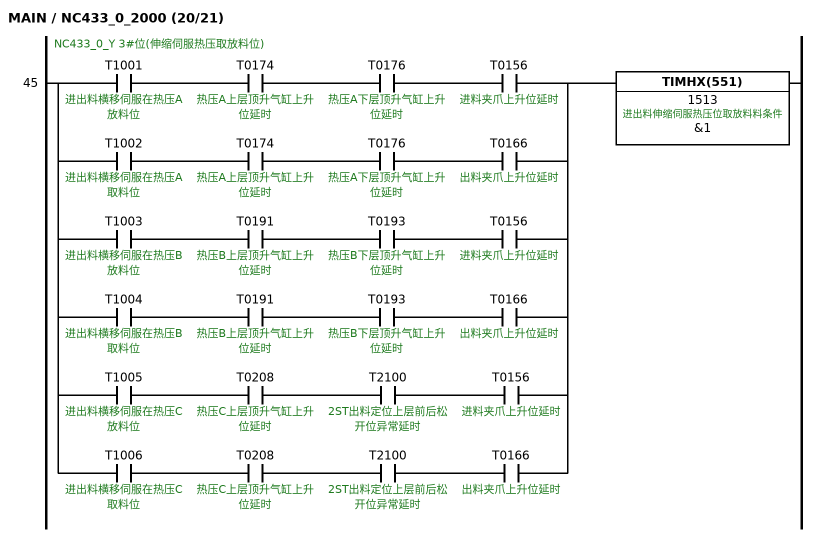
; [picture p24: MAIN / NC433_0_2000, rungs 45-45]
; rung 45: NC433_0_Y 3#位(伸缩伺服热压取放料位)
LD T1001  ; 进出料横移伺服在热压A放料位
AND T0174  ; 热压A上层顶升气缸上升位延时
AND T0176  ; 热压A下层顶升气缸上升位延时
AND T0156  ; 进料夹爪上升位延时
LD T1002  ; 进出料横移伺服在热压A取料位
AND T0174  ; 热压A上层顶升气缸上升位延时
AND T0176  ; 热压A下层顶升气缸上升位延时
AND T0166  ; 出料夹爪上升位延时
ORLD
LD T1003  ; 进出料横移伺服在热压B放料位
AND T0191  ; 热压B上层顶升气缸上升位延时
AND T0193  ; 热压B下层顶升气缸上升位延时
AND T0156  ; 进料夹爪上升位延时
ORLD
LD T1004  ; 进出料横移伺服在热压B取料位
AND T0191  ; 热压B上层顶升气缸上升位延时
AND T0193  ; 热压B下层顶升气缸上升位延时
AND T0166  ; 出料夹爪上升位延时
ORLD
LD T1005  ; 进出料横移伺服在热压C放料位
AND T0208  ; 热压C上层顶升气缸上升位延时
AND T2100  ; 2ST出料定位上层前后松开位异常延时
AND T0156  ; 进料夹爪上升位延时
ORLD
LD T1006  ; 进出料横移伺服在热压C取料位
AND T0208  ; 热压C上层顶升气缸上升位延时
AND T2100  ; 2ST出料定位上层前后松开位异常延时
AND T0166  ; 出料夹爪上升位延时
ORLD
TIMHX(551) 1513 &1  ; 进出料伸缩伺服热压位取放料料条件

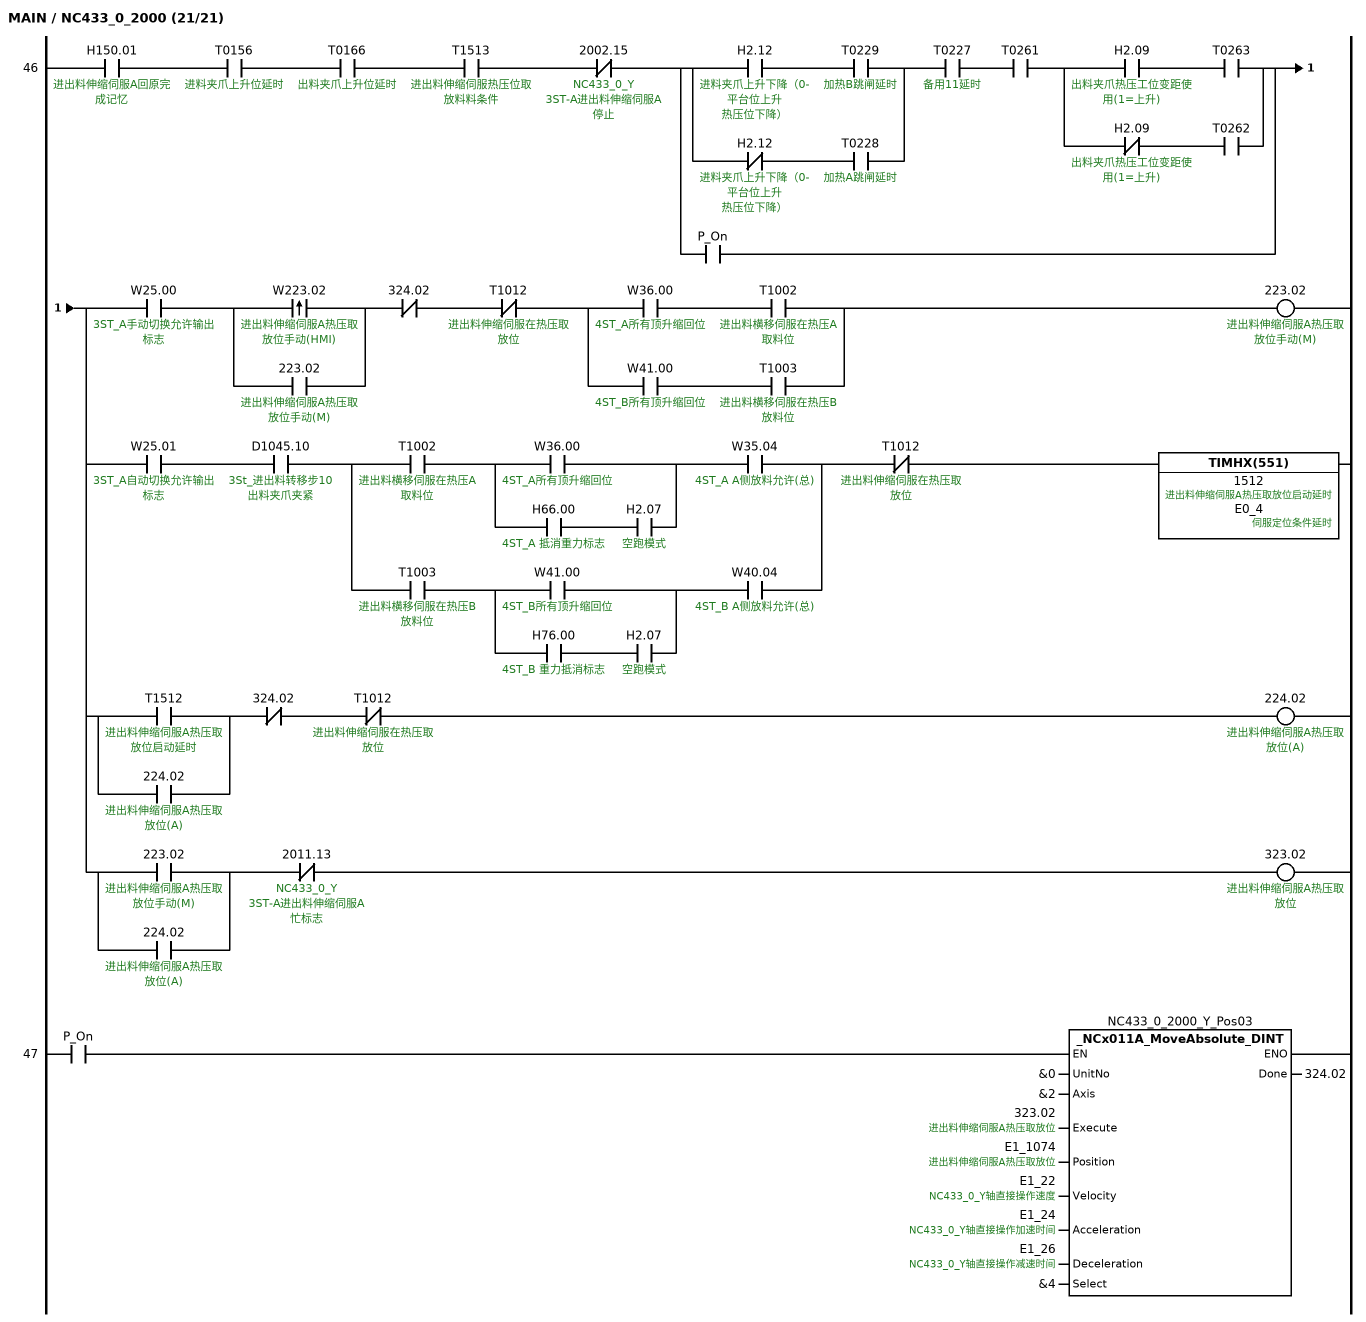
; rung 46
LD H150.01  ; 进出料伸缩伺服A回原完成记忆
AND T0156  ; 进料夹爪上升位延时
AND T0166  ; 出料夹爪上升位延时
AND T1513  ; 进出料伸缩伺服热压位取放料料条件
ANDNOT 2002.15  ; NC433_0_Y 3ST-A进出料伸缩伺服A停止
LD H2.12  ; 进料夹爪上升下降（0-平台位上升  热压位下降）
AND T0229  ; 加热B跳闸延时
LDNOT H2.12  ; 进料夹爪上升下降（0-平台位上升  热压位下降）
AND T0228  ; 加热A跳闸延时
ORLD
AND T0227  ; 备用11延时
AND T0261
LD H2.09  ; 出料夹爪热压工位变距使用(1=上升)
AND T0263
LDNOT H2.09  ; 出料夹爪热压工位变距使用(1=上升)
AND T0262
ORLD
ANDLD
OR P_On
ANDLD
OUT TR0
AND W25.00  ; 3ST_A手动切换允许输出标志
@LD W223.02  ; 进出料伸缩伺服A热压取放位手动(HMI)
OR 223.02  ; 进出料伸缩伺服A热压取放位手动(M)
ANDLD
ANDNOT 324.02
ANDNOT T1012  ; 进出料伸缩伺服在热压取放位
LD W36.00  ; 4ST_A所有顶升缩回位
AND T1002  ; 进出料横移伺服在热压A取料位
LD W41.00  ; 4ST_B所有顶升缩回位
AND T1003  ; 进出料横移伺服在热压B放料位
ORLD
ANDLD
OUT 223.02  ; 进出料伸缩伺服A热压取放位手动(M)
LD TR0
AND W25.01  ; 3ST_A自动切换允许输出标志
AND D1045.10  ; 3St_进出料转移步10 出料夹爪夹紧
LD T1002  ; 进出料横移伺服在热压A取料位
LD W36.00  ; 4ST_A所有顶升缩回位
LD H66.00  ; 4ST_A 抵消重力标志
AND H2.07  ; 空跑模式
ORLD
ANDLD
AND W35.04  ; 4ST_A A侧放料允许(总)
LD T1003  ; 进出料横移伺服在热压B放料位
LD W41.00  ; 4ST_B所有顶升缩回位
LD H76.00  ; 4ST_B 重力抵消标志
AND H2.07  ; 空跑模式
ORLD
ANDLD
AND W40.04  ; 4ST_B A侧放料允许(总)
ORLD
ANDLD
ANDNOT T1012  ; 进出料伸缩伺服在热压取放位
TIMHX(551) 1512 E0_4  ; 伺服定位条件延时, 进出料伸缩伺服A热压取放位启动延时
LD TR0
LD T1512  ; 进出料伸缩伺服A热压取放位启动延时
OR 224.02  ; 进出料伸缩伺服A热压取放位(A)
ANDLD
ANDNOT 324.02
ANDNOT T1012  ; 进出料伸缩伺服在热压取放位
OUT 224.02  ; 进出料伸缩伺服A热压取放位(A)
LD TR0
LD 223.02  ; 进出料伸缩伺服A热压取放位手动(M)
OR 224.02  ; 进出料伸缩伺服A热压取放位(A)
ANDLD
ANDNOT 2011.13  ; NC433_0_Y 3ST-A进出料伸缩伺服A忙标志
OUT 323.02  ; 进出料伸缩伺服A热压取放位
; rung 47
LD P_On
CALL NC433_0_2000_Y_Pos03 : _NCx011A_MoveAbsolute_DINT (UnitNo := &0, Axis := &2, Execute := 323.02, Position := E1_1074, Velocity := E1_22, Acceleration := E1_24, Deceleration := E1_26, Select := &4, Done => 324.02)  ; 进出料伸缩伺服A热压取放位, NC433_0_Y轴直接操作速度, NC433_0_Y轴直接操作加速时间, NC433_0_Y轴直接操作减速时间

### Section 主副PLC交互

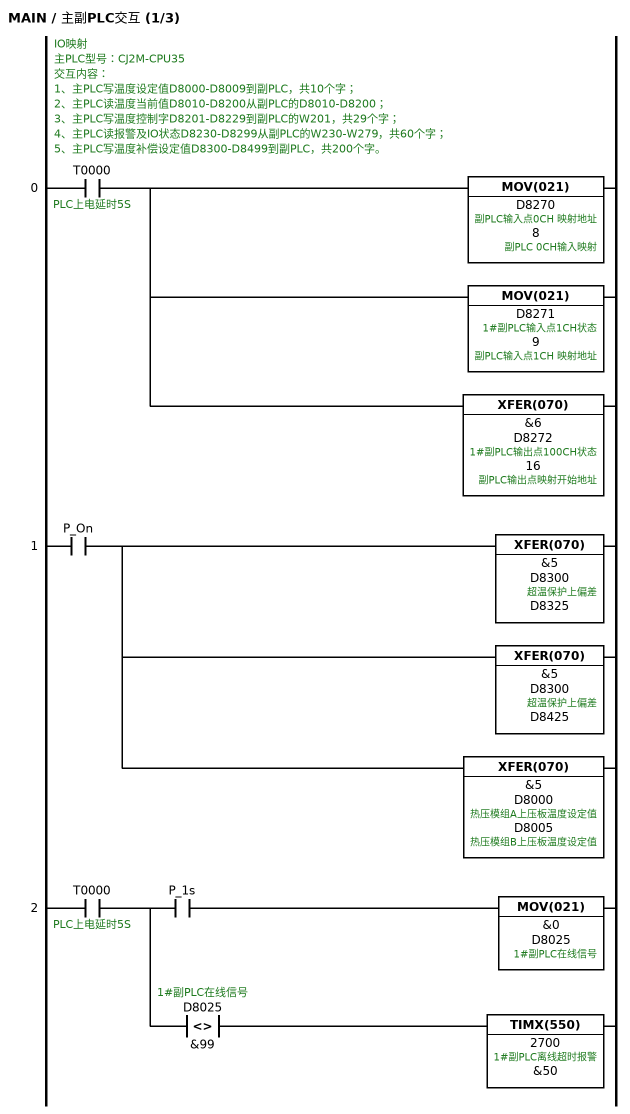
; rung 0: IO映射 / 主PLC型号：CJ2M-CPU35 / 交互内容： / 1、主PLC写温度设定值D8000-D8009到副PLC，共10个字； / 2、主PLC读温度当前值D8010-D8200从副PLC的D8010-D8200； / 3、主PLC写温度控制字D8201-D8229到副PLC的W201，共29个字； / 4、主PLC读报警及IO状态D8230-D8299从副PLC的W230-W279，共60个字； / 5、主PLC写温度补偿设定值D8300-D8499到副PLC，共200个字。
LD T0000  ; PLC上电延时5S
MOV(021) D8270 8  ; 副PLC输入点0CH 映射地址, 副PLC 0CH输入映射
MOV(021) D8271 9  ; 1#副PLC输入点1CH状态, 副PLC输入点1CH 映射地址
XFER(070) &6 D8272 16  ; 1#副PLC输出点100CH状态, 副PLC输出点映射开始地址
; rung 1
LD P_On
XFER(070) &5 D8300 D8325  ; 超温保护上偏差
XFER(070) &5 D8300 D8425  ; 超温保护上偏差
XFER(070) &5 D8000 D8005  ; 热压模组A上压板温度设定值, 热压模组B上压板温度设定值
; rung 2
LD T0000  ; PLC上电延时5S
OUT TR0
AND P_1s
MOV(021) &0 D8025  ; 1#副PLC在线信号
LD TR0
AND<>(305) D8025 &99  ; 1#副PLC在线信号
TIMX(550) 2700 &50  ; 1#副PLC离线超时报警

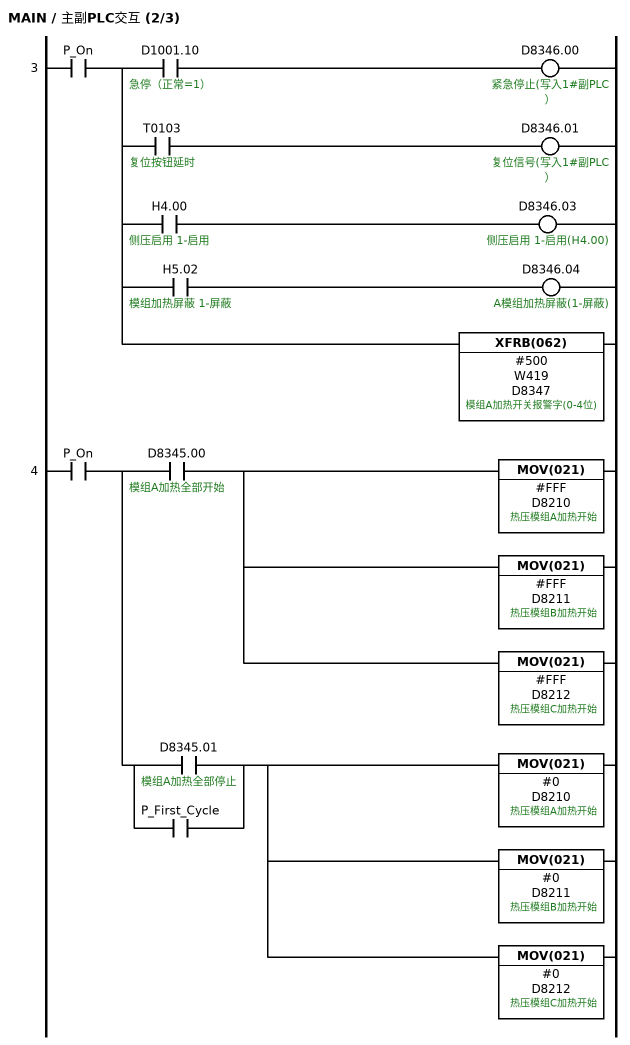
; rung 3
LD P_On
OUT TR0
AND D1001.10  ; 急停（正常=1）
OUT D8346.00  ; 紧急停止(写入1#副PLC）
LD TR0
AND T0103  ; 复位按钮延时
OUT D8346.01  ; 复位信号(写入1#副PLC）
LD TR0
AND H4.00  ; 侧压启用 1-启用
OUT D8346.03  ; 侧压启用 1-启用(H4.00)
LD TR0
AND H5.02  ; 模组加热屏蔽 1-屏蔽
OUT D8346.04  ; A模组加热屏蔽(1-屏蔽)
LD TR0
XFRB(062) #500 W419 D8347  ; 模组A加热开关报警字(0-4位)
; rung 4
LD P_On
OUT TR0
AND D8345.00  ; 模组A加热全部开始
MOV(021) #FFF D8210  ; 热压模组A加热开始
MOV(021) #FFF D8211  ; 热压模组B加热开始
MOV(021) #FFF D8212  ; 热压模组C加热开始
LD TR0
LD D8345.01  ; 模组A加热全部停止
OR P_First_Cycle
ANDLD
MOV(021) #0 D8210  ; 热压模组A加热开始
MOV(021) #0 D8211  ; 热压模组B加热开始
MOV(021) #0 D8212  ; 热压模组C加热开始

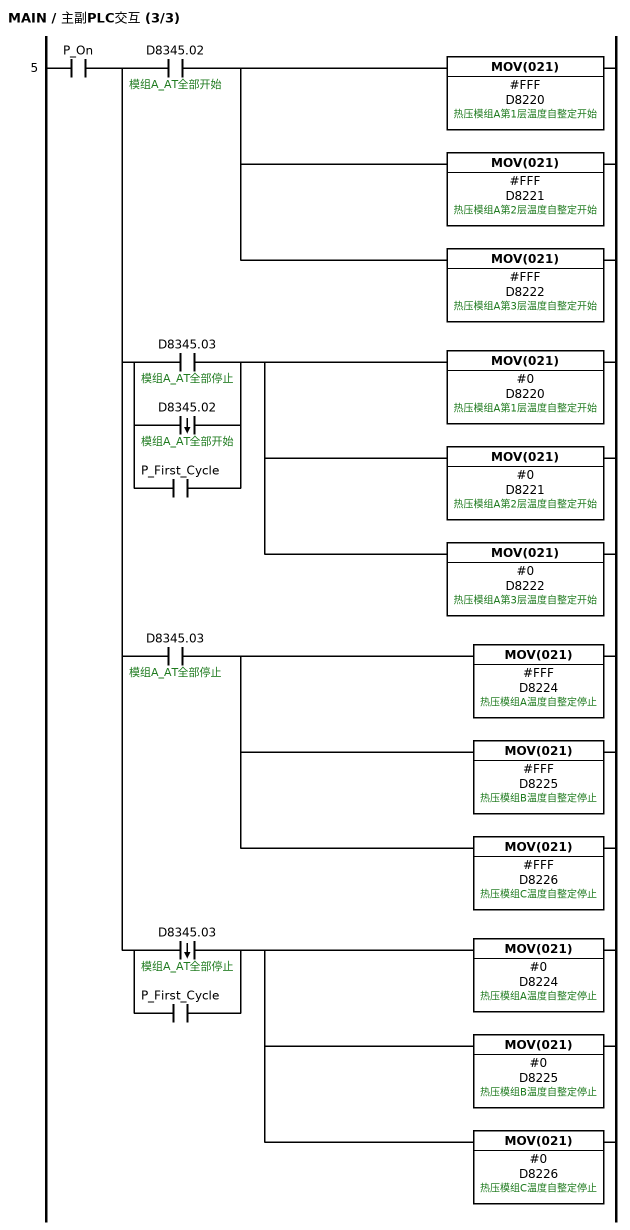
; rung 5
LD P_On
OUT TR0
AND D8345.02  ; 模组A_AT全部开始
MOV(021) #FFF D8220  ; 热压模组A第1层温度自整定开始
MOV(021) #FFF D8221  ; 热压模组A第2层温度自整定开始
MOV(021) #FFF D8222  ; 热压模组A第3层温度自整定开始
LD TR0
LD D8345.03  ; 模组A_AT全部停止
%OR D8345.02  ; 模组A_AT全部开始
OR P_First_Cycle
ANDLD
MOV(021) #0 D8220  ; 热压模组A第1层温度自整定开始
MOV(021) #0 D8221  ; 热压模组A第2层温度自整定开始
MOV(021) #0 D8222  ; 热压模组A第3层温度自整定开始
LD TR0
AND D8345.03  ; 模组A_AT全部停止
MOV(021) #FFF D8224  ; 热压模组A温度自整定停止
MOV(021) #FFF D8225  ; 热压模组B温度自整定停止
MOV(021) #FFF D8226  ; 热压模组C温度自整定停止
LD TR0
%LD D8345.03  ; 模组A_AT全部停止
OR P_First_Cycle
ANDLD
MOV(021) #0 D8224  ; 热压模组A温度自整定停止
MOV(021) #0 D8225  ; 热压模组B温度自整定停止
MOV(021) #0 D8226  ; 热压模组C温度自整定停止

### Section 压力转换

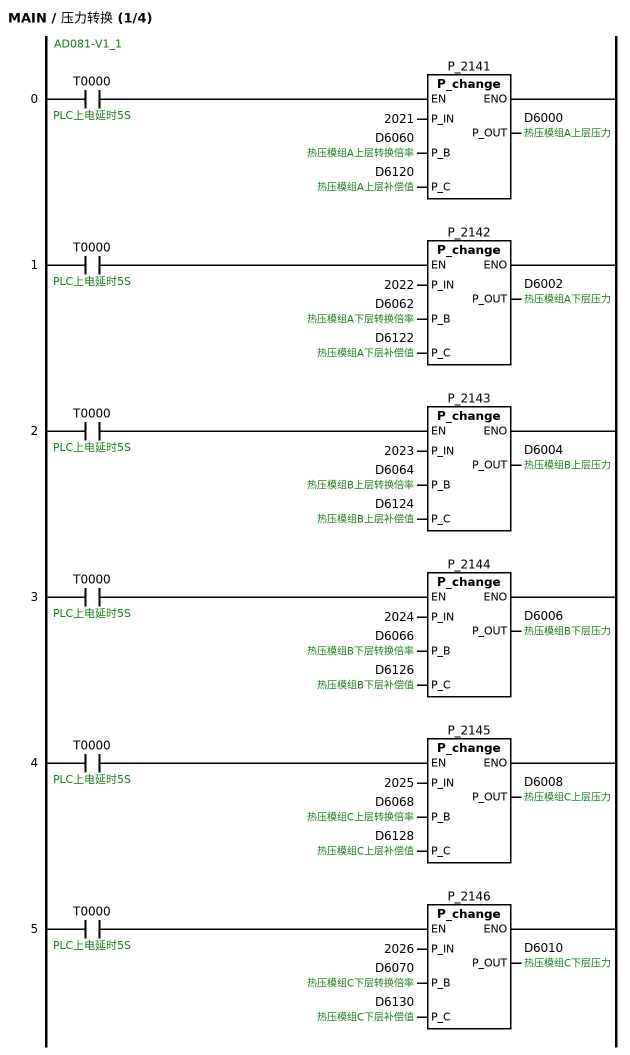
; rung 0: AD081-V1_1
LD T0000  ; PLC上电延时5S
CALL P_2141 : P_change (P_IN := 2021, P_B := D6060, P_C := D6120, P_OUT => D6000)  ; 热压模组A上层转换倍率, 热压模组A上层补偿值, 热压模组A上层压力
; rung 1
LD T0000  ; PLC上电延时5S
CALL P_2142 : P_change (P_IN := 2022, P_B := D6062, P_C := D6122, P_OUT => D6002)  ; 热压模组A下层转换倍率, 热压模组A下层补偿值, 热压模组A下层压力
; rung 2
LD T0000  ; PLC上电延时5S
CALL P_2143 : P_change (P_IN := 2023, P_B := D6064, P_C := D6124, P_OUT => D6004)  ; 热压模组B上层转换倍率, 热压模组B上层补偿值, 热压模组B上层压力
; rung 3
LD T0000  ; PLC上电延时5S
CALL P_2144 : P_change (P_IN := 2024, P_B := D6066, P_C := D6126, P_OUT => D6006)  ; 热压模组B下层转换倍率, 热压模组B下层补偿值, 热压模组B下层压力
; rung 4
LD T0000  ; PLC上电延时5S
CALL P_2145 : P_change (P_IN := 2025, P_B := D6068, P_C := D6128, P_OUT => D6008)  ; 热压模组C上层转换倍率, 热压模组C上层补偿值, 热压模组C上层压力
; rung 5
LD T0000  ; PLC上电延时5S
CALL P_2146 : P_change (P_IN := 2026, P_B := D6070, P_C := D6130, P_OUT => D6010)  ; 热压模组C下层转换倍率, 热压模组C下层补偿值, 热压模组C下层压力

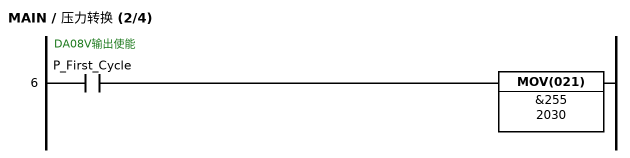
; rung 6: DA08V输出使能
LD P_First_Cycle
MOV(021) &255 2030

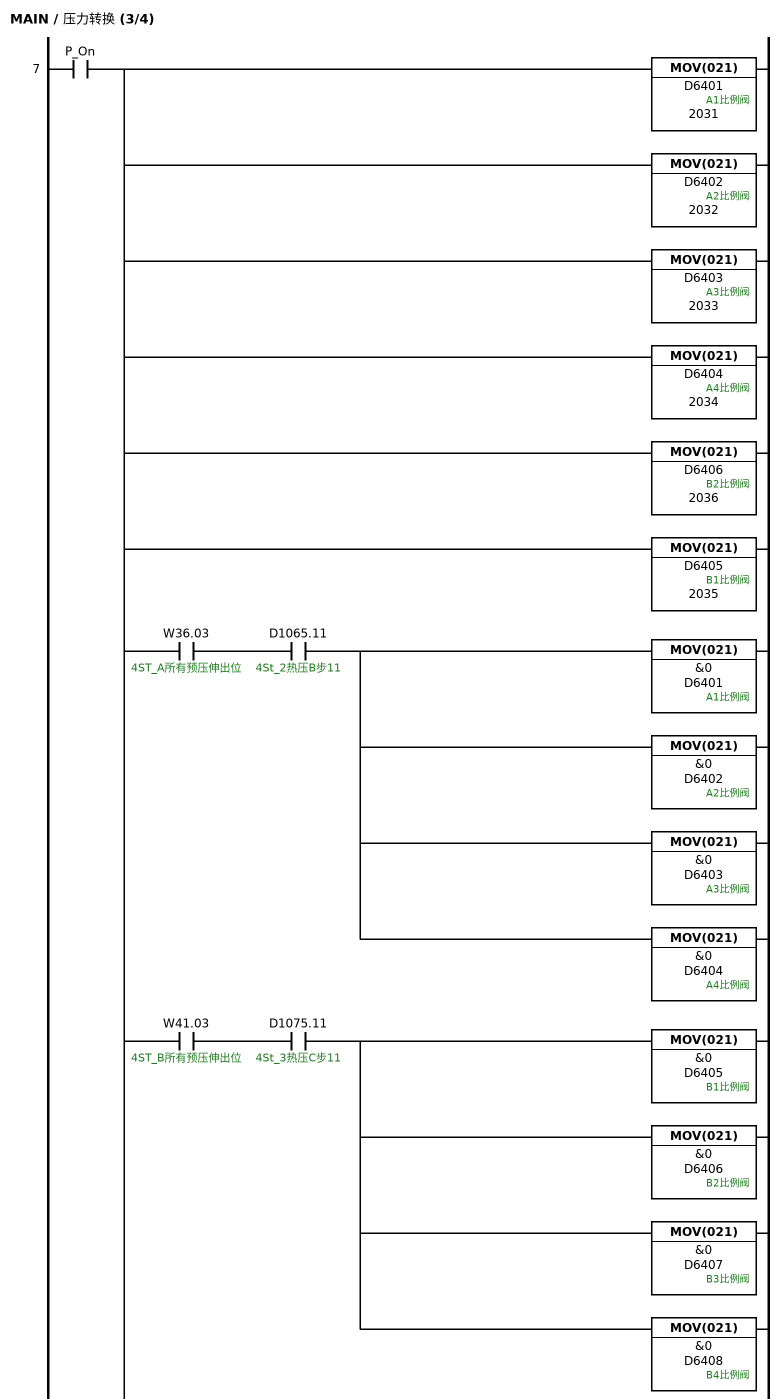

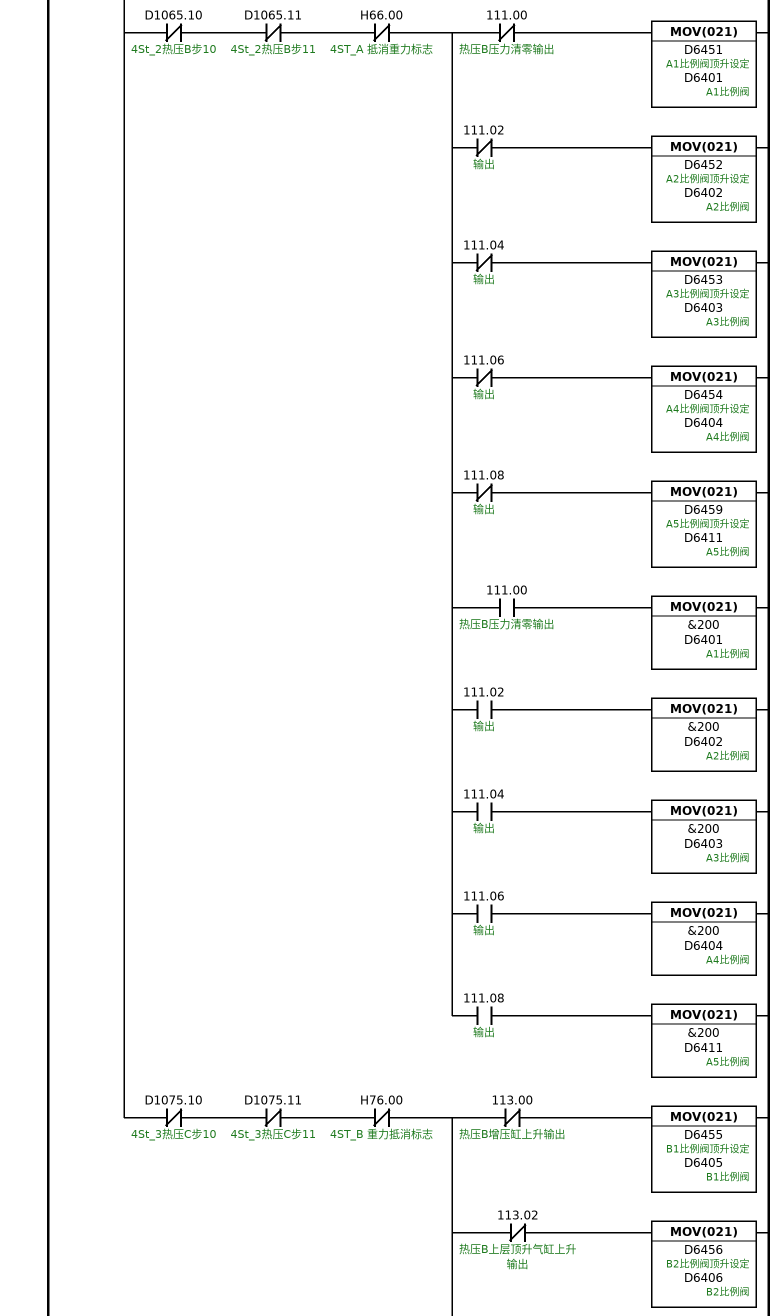

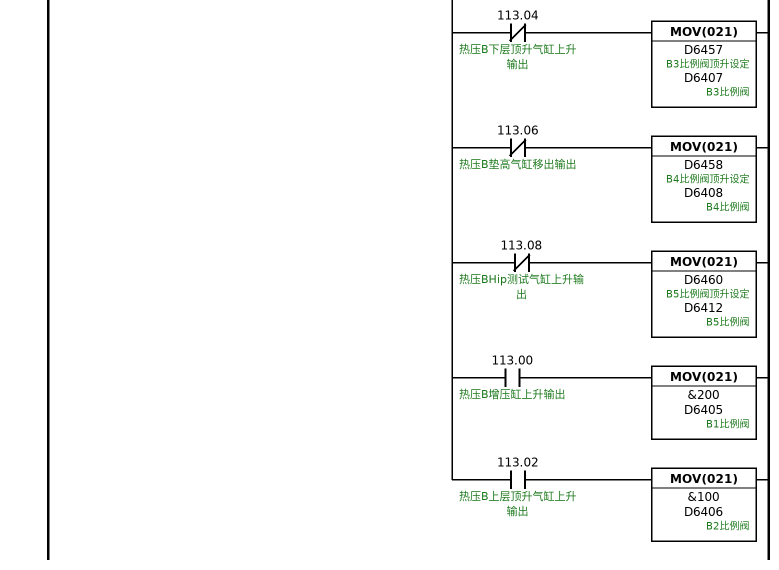
; rung 7
LD P_On
OUT TR0
MOV(021) D6401 2031  ; A1比例阀
MOV(021) D6402 2032  ; A2比例阀
MOV(021) D6403 2033  ; A3比例阀
MOV(021) D6404 2034  ; A4比例阀
MOV(021) D6406 2036  ; B2比例阀
MOV(021) D6405 2035  ; B1比例阀
AND W36.03  ; 4ST_A所有预压伸出位
AND D1065.11  ; 4St_2热压B步11
MOV(021) &0 D6401  ; A1比例阀
MOV(021) &0 D6402  ; A2比例阀
MOV(021) &0 D6403  ; A3比例阀
MOV(021) &0 D6404  ; A4比例阀
LD TR0
AND W41.03  ; 4ST_B所有预压伸出位
AND D1075.11  ; 4St_3热压C步11
MOV(021) &0 D6405  ; B1比例阀
MOV(021) &0 D6406  ; B2比例阀
MOV(021) &0 D6407  ; B3比例阀
MOV(021) &0 D6408  ; B4比例阀
LD TR0
ANDNOT D1065.10  ; 4St_2热压B步10
ANDNOT D1065.11  ; 4St_2热压B步11
ANDNOT H66.00  ; 4ST_A 抵消重力标志
OUT TR1
ANDNOT 111.00  ; 热压B压力清零输出
MOV(021) D6451 D6401  ; A1比例阀顶升设定, A1比例阀
LD TR1
ANDNOT 111.02  ; 输出
MOV(021) D6452 D6402  ; A2比例阀顶升设定, A2比例阀
LD TR1
ANDNOT 111.04  ; 输出
MOV(021) D6453 D6403  ; A3比例阀顶升设定, A3比例阀
LD TR1
ANDNOT 111.06  ; 输出
MOV(021) D6454 D6404  ; A4比例阀顶升设定, A4比例阀
LD TR1
ANDNOT 111.08  ; 输出
MOV(021) D6459 D6411  ; A5比例阀顶升设定, A5比例阀
LD TR1
AND 111.00  ; 热压B压力清零输出
MOV(021) &200 D6401  ; A1比例阀
LD TR1
AND 111.02  ; 输出
MOV(021) &200 D6402  ; A2比例阀
LD TR1
AND 111.04  ; 输出
MOV(021) &200 D6403  ; A3比例阀
LD TR1
AND 111.06  ; 输出
MOV(021) &200 D6404  ; A4比例阀
LD TR1
AND 111.08  ; 输出
MOV(021) &200 D6411  ; A5比例阀
LD TR0
ANDNOT D1075.10  ; 4St_3热压C步10
ANDNOT D1075.11  ; 4St_3热压C步11
ANDNOT H76.00  ; 4ST_B 重力抵消标志
OUT TR0
ANDNOT 113.00  ; 热压B增压缸上升输出
MOV(021) D6455 D6405  ; B1比例阀顶升设定, B1比例阀
LD TR0
ANDNOT 113.02  ; 热压B上层顶升气缸上升输出
MOV(021) D6456 D6406  ; B2比例阀顶升设定, B2比例阀
LD TR0
ANDNOT 113.04  ; 热压B下层顶升气缸上升输出
MOV(021) D6457 D6407  ; B3比例阀顶升设定, B3比例阀
LD TR0
ANDNOT 113.06  ; 热压B垫高气缸移出输出
MOV(021) D6458 D6408  ; B4比例阀顶升设定, B4比例阀
LD TR0
ANDNOT 113.08  ; 热压BHip测试气缸上升输出
MOV(021) D6460 D6412  ; B5比例阀顶升设定, B5比例阀
LD TR0
AND 113.00  ; 热压B增压缸上升输出
MOV(021) &200 D6405  ; B1比例阀
LD TR0
AND 113.02  ; 热压B上层顶升气缸上升输出
MOV(021) &100 D6406  ; B2比例阀

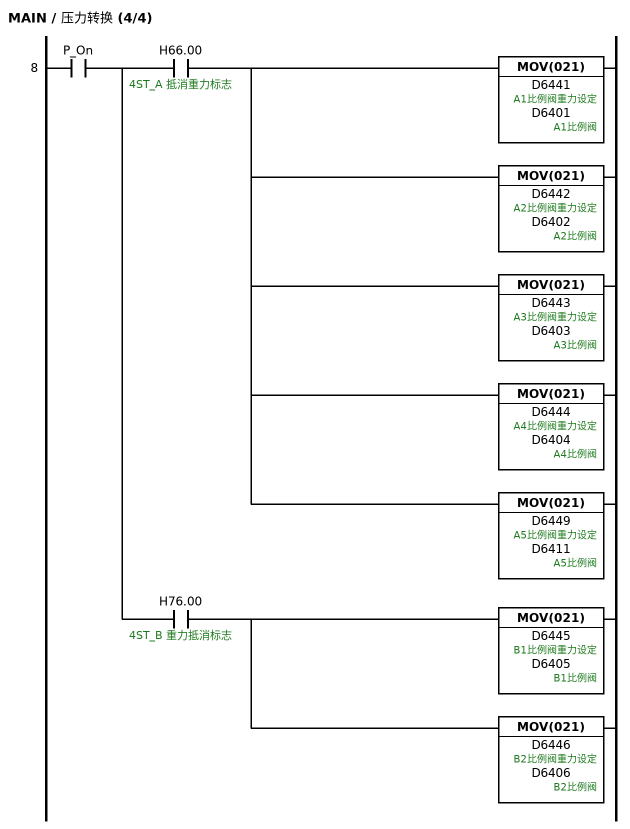
; rung 8
LD P_On
OUT TR0
AND H66.00  ; 4ST_A 抵消重力标志
MOV(021) D6441 D6401  ; A1比例阀重力设定, A1比例阀
MOV(021) D6442 D6402  ; A2比例阀重力设定, A2比例阀
MOV(021) D6443 D6403  ; A3比例阀重力设定, A3比例阀
MOV(021) D6444 D6404  ; A4比例阀重力设定, A4比例阀
MOV(021) D6449 D6411  ; A5比例阀重力设定, A5比例阀
LD TR0
AND H76.00  ; 4ST_B 重力抵消标志
MOV(021) D6445 D6405  ; B1比例阀重力设定, B1比例阀
MOV(021) D6446 D6406  ; B2比例阀重力设定, B2比例阀

### Section 绝缘仪
; SCU21_3 Port#1:ST5520 通讯协议：38400,8,1,N。

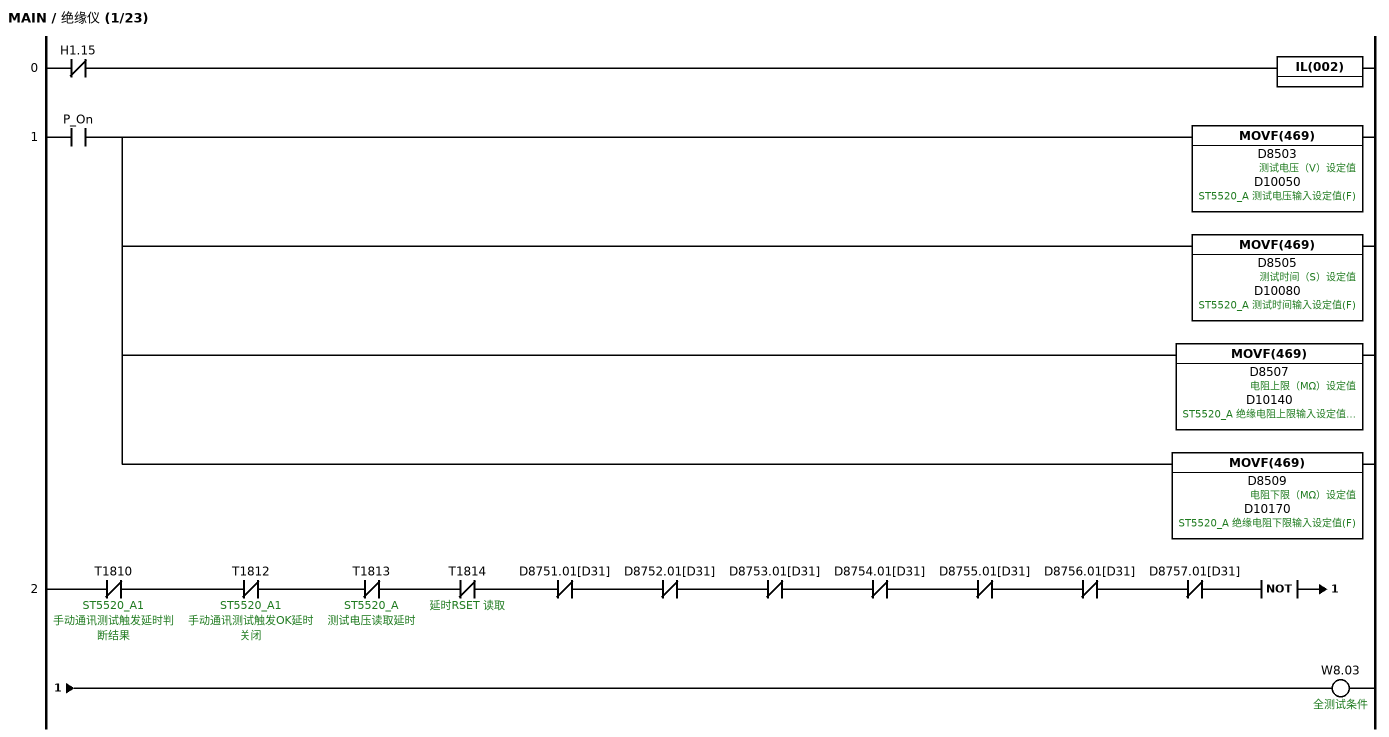
; rung 0
LDNOT H1.15
IL(002)
; rung 1
LD P_On
MOVF(469) D8503 D10050  ; 测试电压（V）设定值, ST5520_A 测试电压输入设定值(F)
MOVF(469) D8505 D10080  ; 测试时间（S）设定值, ST5520_A 测试时间输入设定值(F)
MOVF(469) D8507 D10140  ; 电阻上限（MΩ）设定值, ST5520_A 绝缘电阻上限输入设定值(Float)
MOVF(469) D8509 D10170  ; 电阻下限（MΩ）设定值, ST5520_A 绝缘电阻下限输入设定值(F)
; rung 2
LDNOT T1810  ; ST5520_A1 手动通讯测试触发延时判断结果
ANDNOT T1812  ; ST5520_A1 手动通讯测试触发OK延时关闭
ANDNOT T1813  ; ST5520_A 测试电压读取延时
ANDNOT T1814  ; 延时RSET 读取
ANDNOT D8751.01[D31]
ANDNOT D8752.01[D31]
ANDNOT D8753.01[D31]
ANDNOT D8754.01[D31]
ANDNOT D8755.01[D31]
ANDNOT D8756.01[D31]
ANDNOT D8757.01[D31]
NOT(520)
OUT W8.03  ; 全测试条件

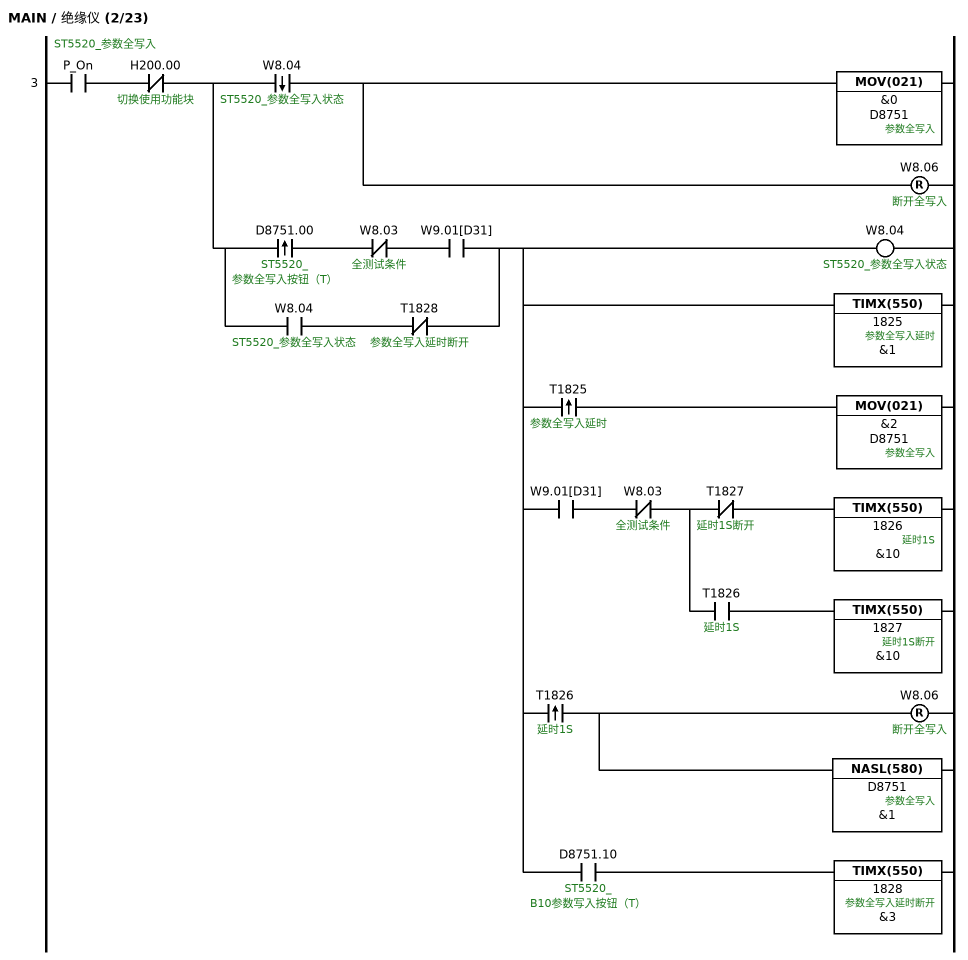
; rung 3: ST5520_参数全写入
LD P_On
ANDNOT H200.00  ; 切换使用功能块
OUT TR0
%AND W8.04  ; ST5520_参数全写入状态
MOV(021) &0 D8751  ; 参数全写入
RSET W8.06  ; 断开全写入
LD TR0
@LD D8751.00  ; ST5520_参数全写入按钮（T）
ANDNOT W8.03  ; 全测试条件
AND W9.01[D31]
LD W8.04  ; ST5520_参数全写入状态
ANDNOT T1828  ; 参数全写入延时断开
ORLD
ANDLD
OUT TR0
OUT W8.04  ; ST5520_参数全写入状态
TIMX(550) 1825 &1  ; 参数全写入延时
@AND T1825  ; 参数全写入延时
MOV(021) &2 D8751  ; 参数全写入
LD TR0
AND W9.01[D31]
ANDNOT W8.03  ; 全测试条件
OUT TR1
ANDNOT T1827  ; 延时1S断开
TIMX(550) 1826 &10  ; 延时1S
LD TR1
AND T1826  ; 延时1S
TIMX(550) 1827 &10  ; 延时1S断开
LD TR0
@AND T1826  ; 延时1S
RSET W8.06  ; 断开全写入
NASL(580) D8751 &1  ; 参数全写入
LD TR0
AND D8751.10  ; ST5520_B10参数写入按钮（T）
TIMX(550) 1828 &3  ; 参数全写入延时断开

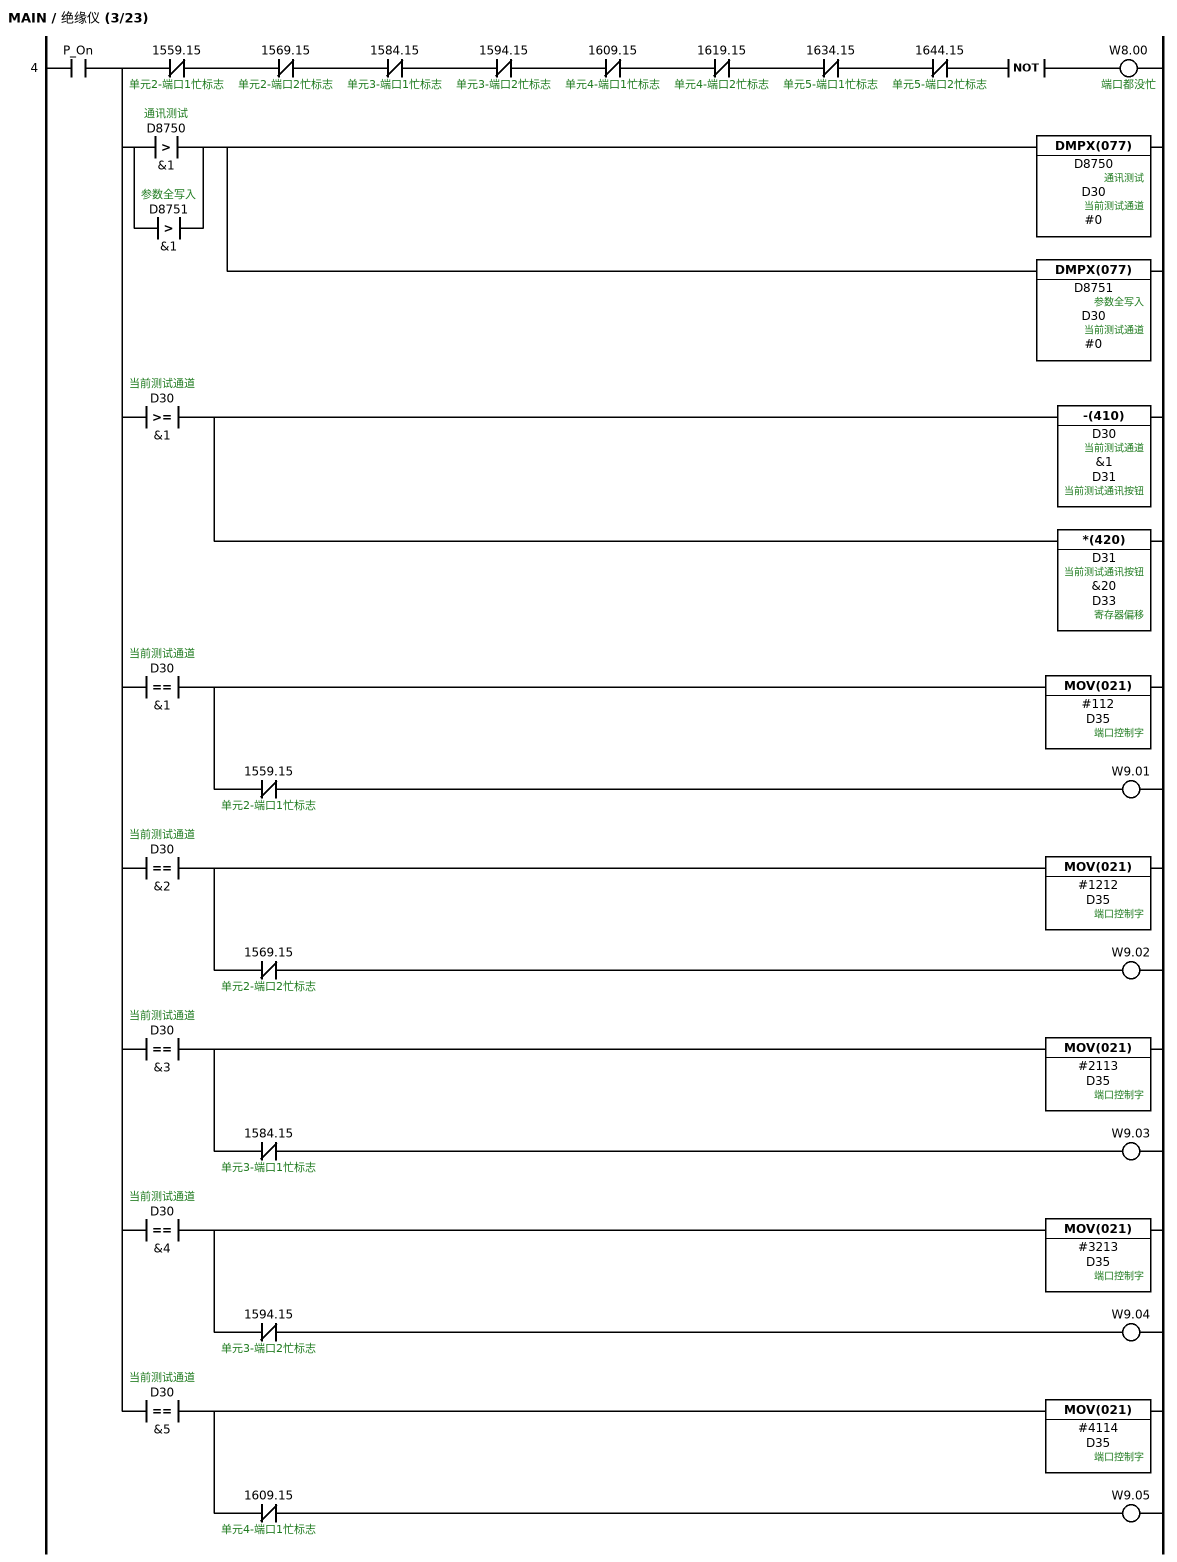
; rung 4
LD P_On
OUT TR0
ANDNOT 1559.15  ; 单元2-端口1忙标志
ANDNOT 1569.15  ; 单元2-端口2忙标志
ANDNOT 1584.15  ; 单元3-端口1忙标志
ANDNOT 1594.15  ; 单元3-端口2忙标志
ANDNOT 1609.15  ; 单元4-端口1忙标志
ANDNOT 1619.15  ; 单元4-端口2忙标志
ANDNOT 1634.15  ; 单元5-端口1忙标志
ANDNOT 1644.15  ; 单元5-端口2忙标志
NOT(520)
OUT W8.00  ; 端口都没忙
LD TR0
LD>(320) D8750 &1  ; 通讯测试
OR>(320) D8751 &1  ; 参数全写入
ANDLD
DMPX(077) D8750 D30 #0  ; 通讯测试, 当前测试通道
DMPX(077) D8751 D30 #0  ; 参数全写入, 当前测试通道
LD TR0
AND>=(325) D30 &1  ; 当前测试通道
-(410) D30 &1 D31  ; 当前测试通道, 当前测试通讯按钮
*(420) D31 &20 D33  ; 当前测试通讯按钮, 寄存器偏移
LD TR0
AND=(300) D30 &1  ; 当前测试通道
MOV(021) #112 D35  ; 端口控制字
ANDNOT 1559.15  ; 单元2-端口1忙标志
OUT W9.01
LD TR0
AND=(300) D30 &2  ; 当前测试通道
MOV(021) #1212 D35  ; 端口控制字
ANDNOT 1569.15  ; 单元2-端口2忙标志
OUT W9.02
LD TR0
AND=(300) D30 &3  ; 当前测试通道
MOV(021) #2113 D35  ; 端口控制字
ANDNOT 1584.15  ; 单元3-端口1忙标志
OUT W9.03
LD TR0
AND=(300) D30 &4  ; 当前测试通道
MOV(021) #3213 D35  ; 端口控制字
ANDNOT 1594.15  ; 单元3-端口2忙标志
OUT W9.04
LD TR0
AND=(300) D30 &5  ; 当前测试通道
MOV(021) #4114 D35  ; 端口控制字
ANDNOT 1609.15  ; 单元4-端口1忙标志
OUT W9.05

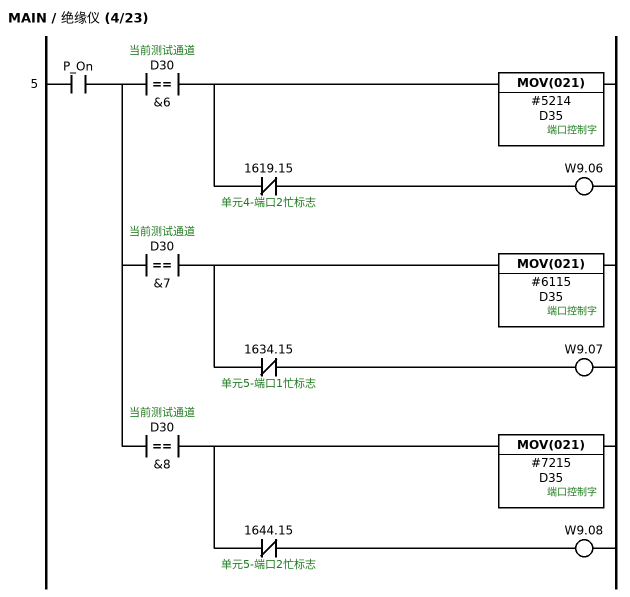
; rung 5
LD P_On
OUT TR0
AND=(300) D30 &6  ; 当前测试通道
MOV(021) #5214 D35  ; 端口控制字
ANDNOT 1619.15  ; 单元4-端口2忙标志
OUT W9.06
LD TR0
AND=(300) D30 &7  ; 当前测试通道
MOV(021) #6115 D35  ; 端口控制字
ANDNOT 1634.15  ; 单元5-端口1忙标志
OUT W9.07
LD TR0
AND=(300) D30 &8  ; 当前测试通道
MOV(021) #7215 D35  ; 端口控制字
ANDNOT 1644.15  ; 单元5-端口2忙标志
OUT W9.08

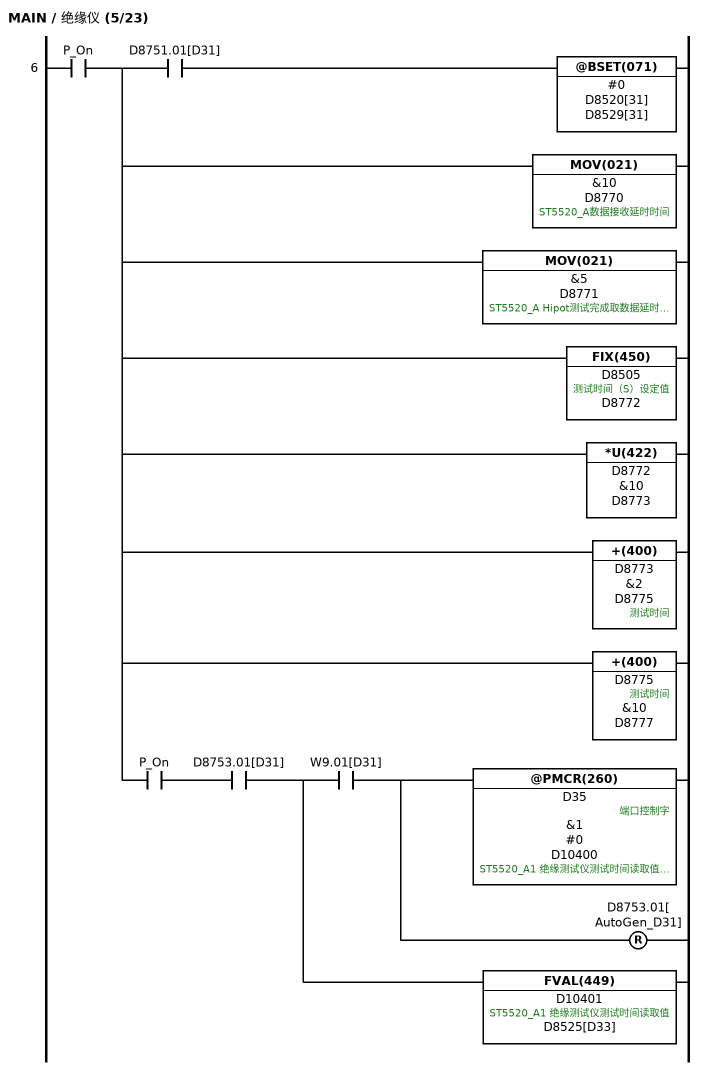
; rung 6
LD P_On
OUT TR0
AND D8751.01[D31]
@BSET(071) #0 D8520[31] D8529[31]
LD TR0
MOV(021) &10 D8770  ; ST5520_A数据接收延时时间
MOV(021) &5 D8771  ; ST5520_A Hipot测试完成取数据延时设定
FIX(450) D8505 D8772  ; 测试时间（S）设定值
*U(422) D8772 &10 D8773
+(400) D8773 &2 D8775  ; 测试时间
+(400) D8775 &10 D8777  ; 测试时间
AND P_On
AND D8753.01[D31]
OUT TR0
AND W9.01[D31]
@PMCR(260) D35 &1 #0 D10400  ; 端口控制字, ST5520_A1 绝缘测试仪测试时间读取值(ASC)
RSET D8753.01[AutoGen_D31]
LD TR0
FVAL(449) D10401 D8525[D33]  ; ST5520_A1 绝缘测试仪测试时间读取值

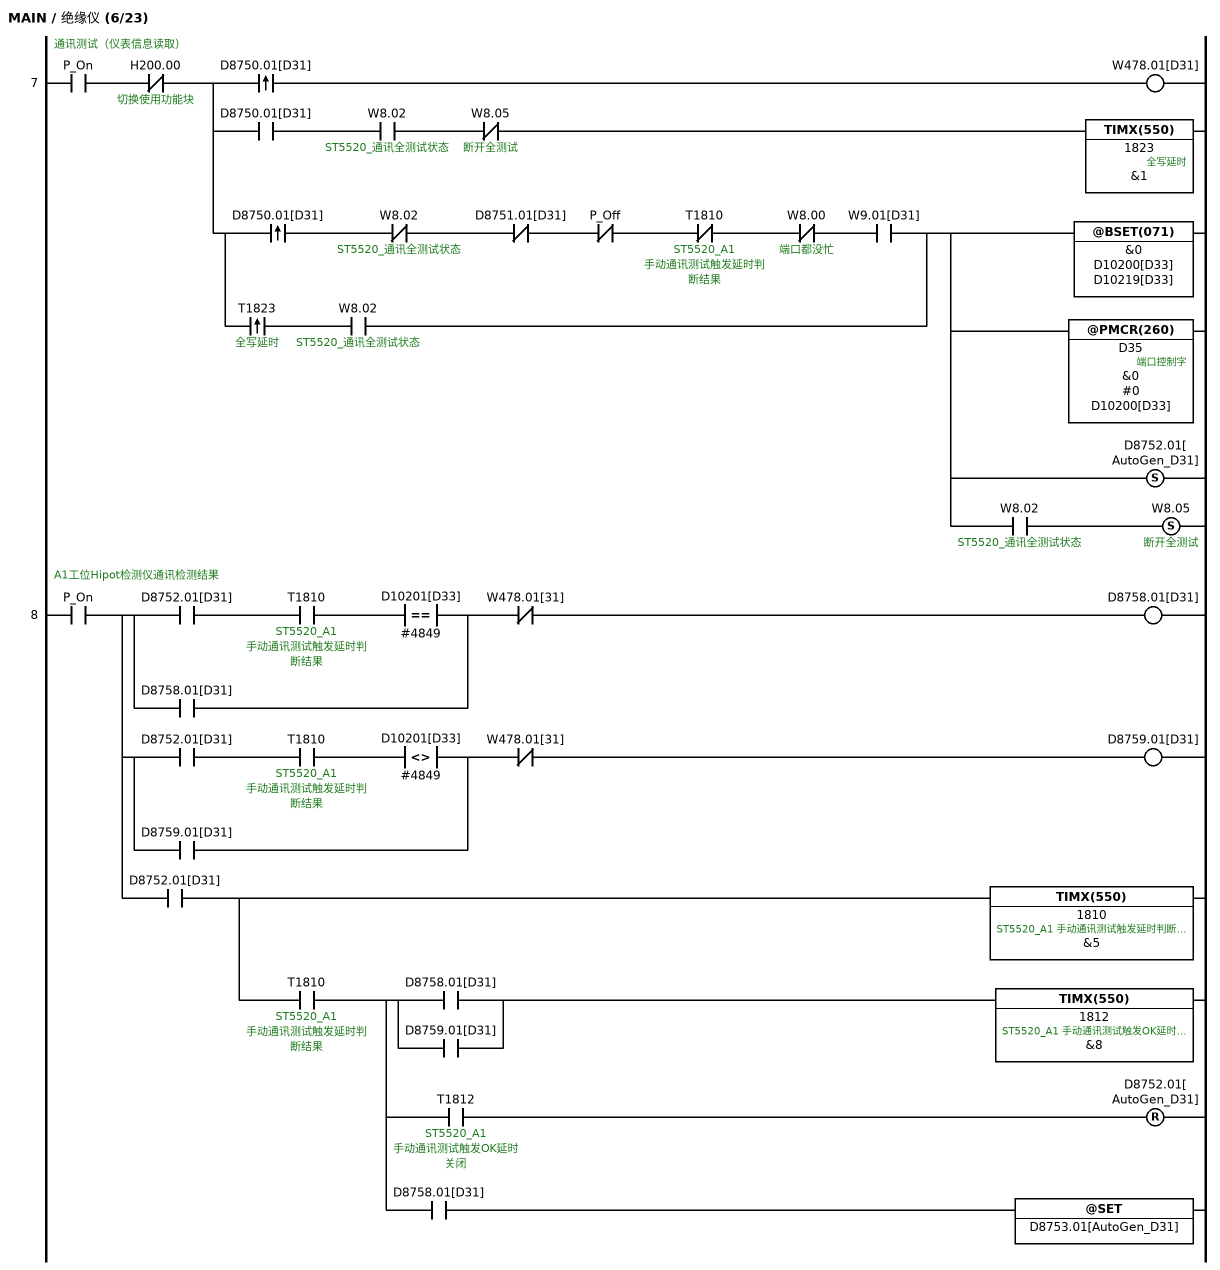
; rung 7: 通讯测试（仪表信息读取）
LD P_On
ANDNOT H200.00  ; 切换使用功能块
OUT TR0
@AND D8750.01[D31]
OUT W478.01[D31]
LD TR0
AND D8750.01[D31]
AND W8.02  ; ST5520_通讯全测试状态
ANDNOT W8.05  ; 断开全测试
TIMX(550) 1823 &1  ; 全写延时
LD TR0
@LD D8750.01[D31]
ANDNOT W8.02  ; ST5520_通讯全测试状态
ANDNOT D8751.01[D31]
ANDNOT P_Off
ANDNOT T1810  ; ST5520_A1 手动通讯测试触发延时判断结果
ANDNOT W8.00  ; 端口都没忙
AND W9.01[D31]
@LD T1823  ; 全写延时
AND W8.02  ; ST5520_通讯全测试状态
ORLD
ANDLD
@BSET(071) &0 D10200[D33] D10219[D33]
@PMCR(260) D35 &0 #0 D10200[D33]  ; 端口控制字
SET D8752.01[AutoGen_D31]
AND W8.02  ; ST5520_通讯全测试状态
SET W8.05  ; 断开全测试
; rung 8: A1工位Hipot检测仪通讯检测结果
LD P_On
OUT TR0
LD D8752.01[D31]
AND T1810  ; ST5520_A1 手动通讯测试触发延时判断结果
AND=(300) D10201[D33] #4849
OR D8758.01[D31]
ANDLD
ANDNOT W478.01[31]
OUT D8758.01[D31]
LD TR0
LD D8752.01[D31]
AND T1810  ; ST5520_A1 手动通讯测试触发延时判断结果
AND<>(305) D10201[D33] #4849
OR D8759.01[D31]
ANDLD
ANDNOT W478.01[31]
OUT D8759.01[D31]
LD TR0
AND D8752.01[D31]
TIMX(550) 1810 &5  ; ST5520_A1 手动通讯测试触发延时判断结果
AND T1810  ; ST5520_A1 手动通讯测试触发延时判断结果
OUT TR0
LD D8758.01[D31]
OR D8759.01[D31]
ANDLD
TIMX(550) 1812 &8  ; ST5520_A1 手动通讯测试触发OK延时关闭
LD TR0
AND T1812  ; ST5520_A1 手动通讯测试触发OK延时关闭
RSET D8752.01[AutoGen_D31]
LD TR0
AND D8758.01[D31]
@SET D8753.01[AutoGen_D31]

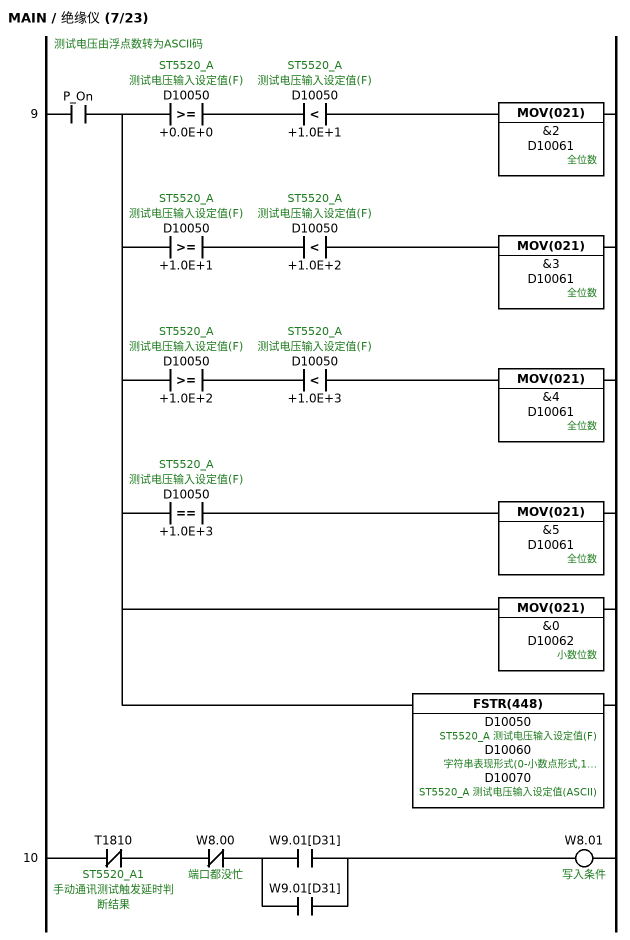
; rung 9: 测试电压由浮点数转为ASCII码
LD P_On
OUT TR0
AND>=F(334) D10050 +0.0E+0  ; ST5520_A 测试电压输入设定值(F)
AND<F(331) D10050 +1.0E+1  ; ST5520_A 测试电压输入设定值(F)
MOV(021) &2 D10061  ; 全位数
LD TR0
AND>=F(334) D10050 +1.0E+1  ; ST5520_A 测试电压输入设定值(F)
AND<F(331) D10050 +1.0E+2  ; ST5520_A 测试电压输入设定值(F)
MOV(021) &3 D10061  ; 全位数
LD TR0
AND>=F(334) D10050 +1.0E+2  ; ST5520_A 测试电压输入设定值(F)
AND<F(331) D10050 +1.0E+3  ; ST5520_A 测试电压输入设定值(F)
MOV(021) &4 D10061  ; 全位数
LD TR0
AND=F(329) D10050 +1.0E+3  ; ST5520_A 测试电压输入设定值(F)
MOV(021) &5 D10061  ; 全位数
LD TR0
MOV(021) &0 D10062  ; 小数位数
FSTR(448) D10050 D10060 D10070  ; ST5520_A 测试电压输入设定值(F), 字符串表现形式(0-小数点形式,1-指数形式), ST5520_A 测试电压输入设定值(ASCII)
; rung 10
LDNOT T1810  ; ST5520_A1 手动通讯测试触发延时判断结果
ANDNOT W8.00  ; 端口都没忙
LD W9.01[D31]
OR W9.01[D31]
ANDLD
OUT W8.01  ; 写入条件

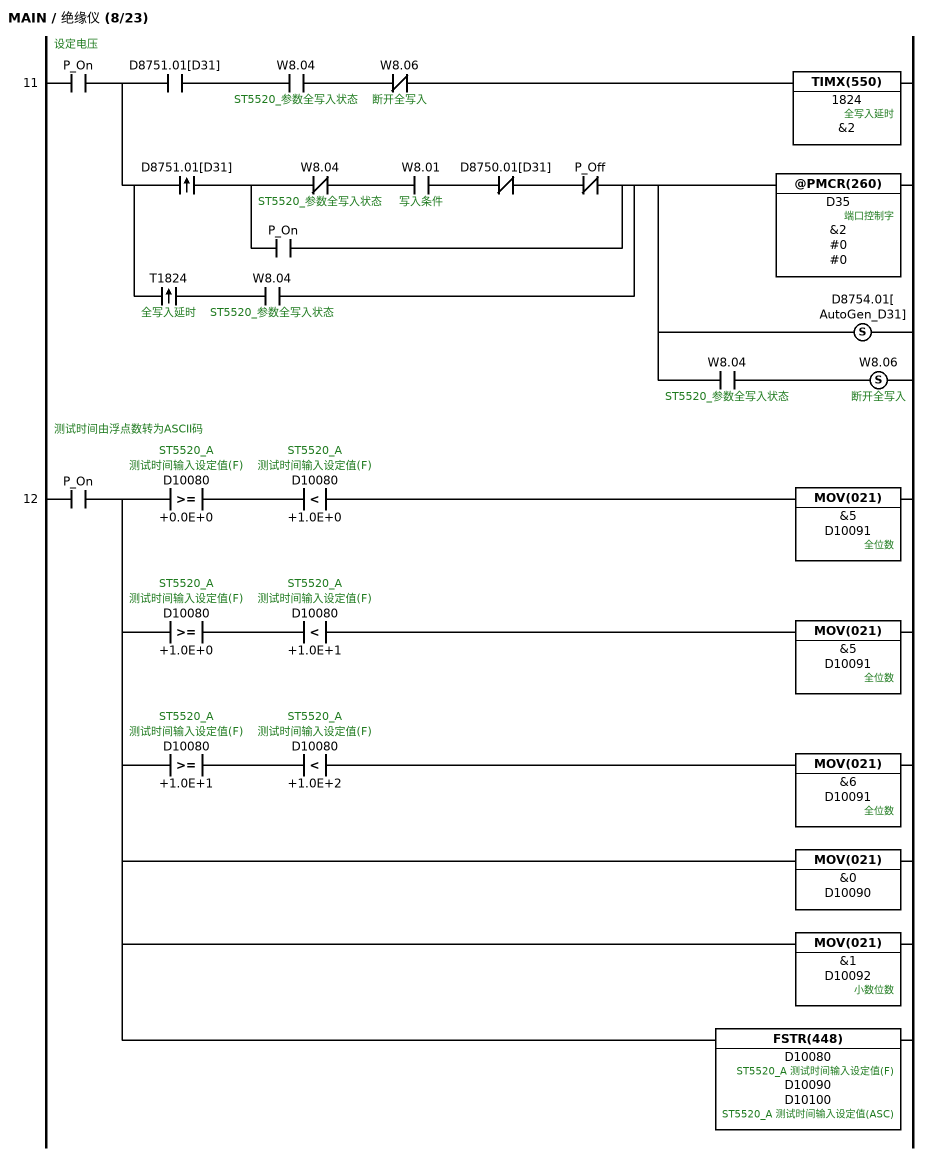
; rung 11: 设定电压
LD P_On
OUT TR0
AND D8751.01[D31]
AND W8.04  ; ST5520_参数全写入状态
ANDNOT W8.06  ; 断开全写入
TIMX(550) 1824 &2  ; 全写入延时
LD TR0
@LD D8751.01[D31]
LDNOT W8.04  ; ST5520_参数全写入状态
AND W8.01  ; 写入条件
ANDNOT D8750.01[D31]
ANDNOT P_Off
OR P_On
ANDLD
@LD T1824  ; 全写入延时
AND W8.04  ; ST5520_参数全写入状态
ORLD
ANDLD
@PMCR(260) D35 &2 #0 #0  ; 端口控制字
SET D8754.01[AutoGen_D31]
AND W8.04  ; ST5520_参数全写入状态
SET W8.06  ; 断开全写入
; rung 12: 测试时间由浮点数转为ASCII码
LD P_On
OUT TR0
AND>=F(334) D10080 +0.0E+0  ; ST5520_A 测试时间输入设定值(F)
AND<F(331) D10080 +1.0E+0  ; ST5520_A 测试时间输入设定值(F)
MOV(021) &5 D10091  ; 全位数
LD TR0
AND>=F(334) D10080 +1.0E+0  ; ST5520_A 测试时间输入设定值(F)
AND<F(331) D10080 +1.0E+1  ; ST5520_A 测试时间输入设定值(F)
MOV(021) &5 D10091  ; 全位数
LD TR0
AND>=F(334) D10080 +1.0E+1  ; ST5520_A 测试时间输入设定值(F)
AND<F(331) D10080 +1.0E+2  ; ST5520_A 测试时间输入设定值(F)
MOV(021) &6 D10091  ; 全位数
LD TR0
MOV(021) &0 D10090
MOV(021) &1 D10092  ; 小数位数
FSTR(448) D10080 D10090 D10100  ; ST5520_A 测试时间输入设定值(F), ST5520_A 测试时间输入设定值(ASC)

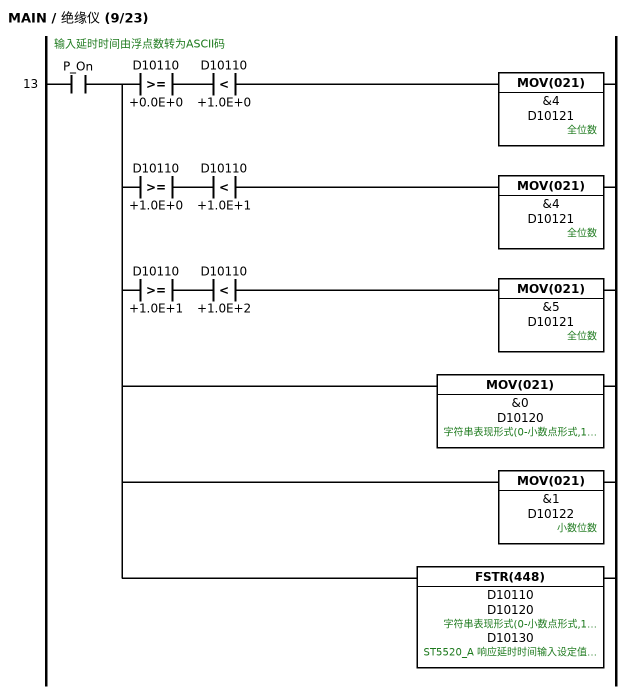
; rung 13: 输入延时时间由浮点数转为ASCII码
LD P_On
OUT TR0
AND>=F(334) D10110 +0.0E+0
AND<F(331) D10110 +1.0E+0
MOV(021) &4 D10121  ; 全位数
LD TR0
AND>=F(334) D10110 +1.0E+0
AND<F(331) D10110 +1.0E+1
MOV(021) &4 D10121  ; 全位数
LD TR0
AND>=F(334) D10110 +1.0E+1
AND<F(331) D10110 +1.0E+2
MOV(021) &5 D10121  ; 全位数
LD TR0
MOV(021) &0 D10120  ; 字符串表现形式(0-小数点形式,1-指数形式)
MOV(021) &1 D10122  ; 小数位数
FSTR(448) D10110 D10120 D10130  ; 字符串表现形式(0-小数点形式,1-指数形式), ST5520_A 响应延时时间输入设定值(ASC)

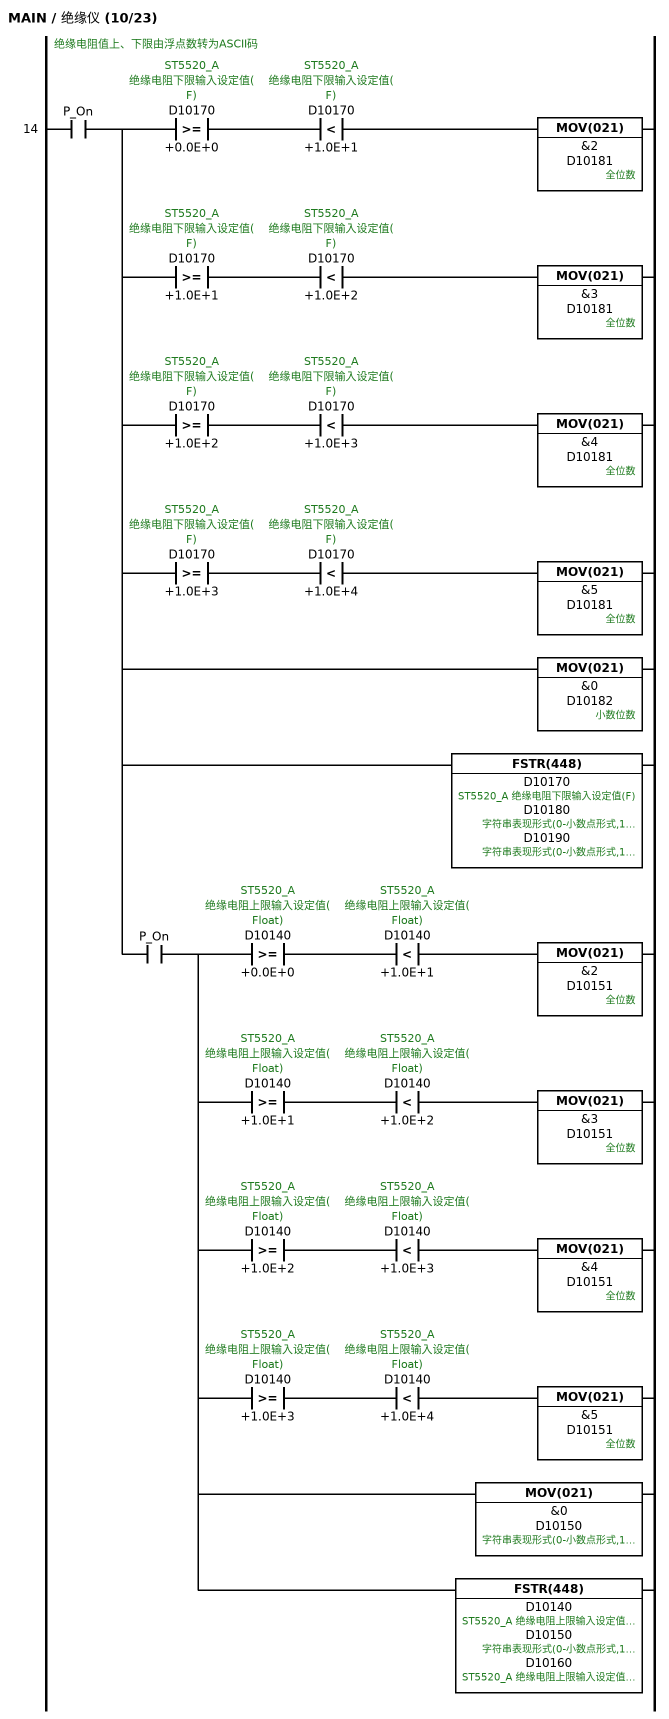
; rung 14: 绝缘电阻值上、下限由浮点数转为ASCII码
LD P_On
OUT TR0
AND>=F(334) D10170 +0.0E+0  ; ST5520_A 绝缘电阻下限输入设定值(F)
AND<F(331) D10170 +1.0E+1  ; ST5520_A 绝缘电阻下限输入设定值(F)
MOV(021) &2 D10181  ; 全位数
LD TR0
AND>=F(334) D10170 +1.0E+1  ; ST5520_A 绝缘电阻下限输入设定值(F)
AND<F(331) D10170 +1.0E+2  ; ST5520_A 绝缘电阻下限输入设定值(F)
MOV(021) &3 D10181  ; 全位数
LD TR0
AND>=F(334) D10170 +1.0E+2  ; ST5520_A 绝缘电阻下限输入设定值(F)
AND<F(331) D10170 +1.0E+3  ; ST5520_A 绝缘电阻下限输入设定值(F)
MOV(021) &4 D10181  ; 全位数
LD TR0
AND>=F(334) D10170 +1.0E+3  ; ST5520_A 绝缘电阻下限输入设定值(F)
AND<F(331) D10170 +1.0E+4  ; ST5520_A 绝缘电阻下限输入设定值(F)
MOV(021) &5 D10181  ; 全位数
LD TR0
MOV(021) &0 D10182  ; 小数位数
FSTR(448) D10170 D10180 D10190  ; ST5520_A 绝缘电阻下限输入设定值(F), 字符串表现形式(0-小数点形式,1-指数形式)
AND P_On
OUT TR0
AND>=F(334) D10140 +0.0E+0  ; ST5520_A 绝缘电阻上限输入设定值(Float)
AND<F(331) D10140 +1.0E+1  ; ST5520_A 绝缘电阻上限输入设定值(Float)
MOV(021) &2 D10151  ; 全位数
LD TR0
AND>=F(334) D10140 +1.0E+1  ; ST5520_A 绝缘电阻上限输入设定值(Float)
AND<F(331) D10140 +1.0E+2  ; ST5520_A 绝缘电阻上限输入设定值(Float)
MOV(021) &3 D10151  ; 全位数
LD TR0
AND>=F(334) D10140 +1.0E+2  ; ST5520_A 绝缘电阻上限输入设定值(Float)
AND<F(331) D10140 +1.0E+3  ; ST5520_A 绝缘电阻上限输入设定值(Float)
MOV(021) &4 D10151  ; 全位数
LD TR0
AND>=F(334) D10140 +1.0E+3  ; ST5520_A 绝缘电阻上限输入设定值(Float)
AND<F(331) D10140 +1.0E+4  ; ST5520_A 绝缘电阻上限输入设定值(Float)
MOV(021) &5 D10151  ; 全位数
LD TR0
MOV(021) &0 D10150  ; 字符串表现形式(0-小数点形式,1-指数形式)
FSTR(448) D10140 D10150 D10160  ; ST5520_A 绝缘电阻上限输入设定值(Float), 字符串表现形式(0-小数点形式,1-指数形式), ST5520_A 绝缘电阻上限输入设定值(ASCII)

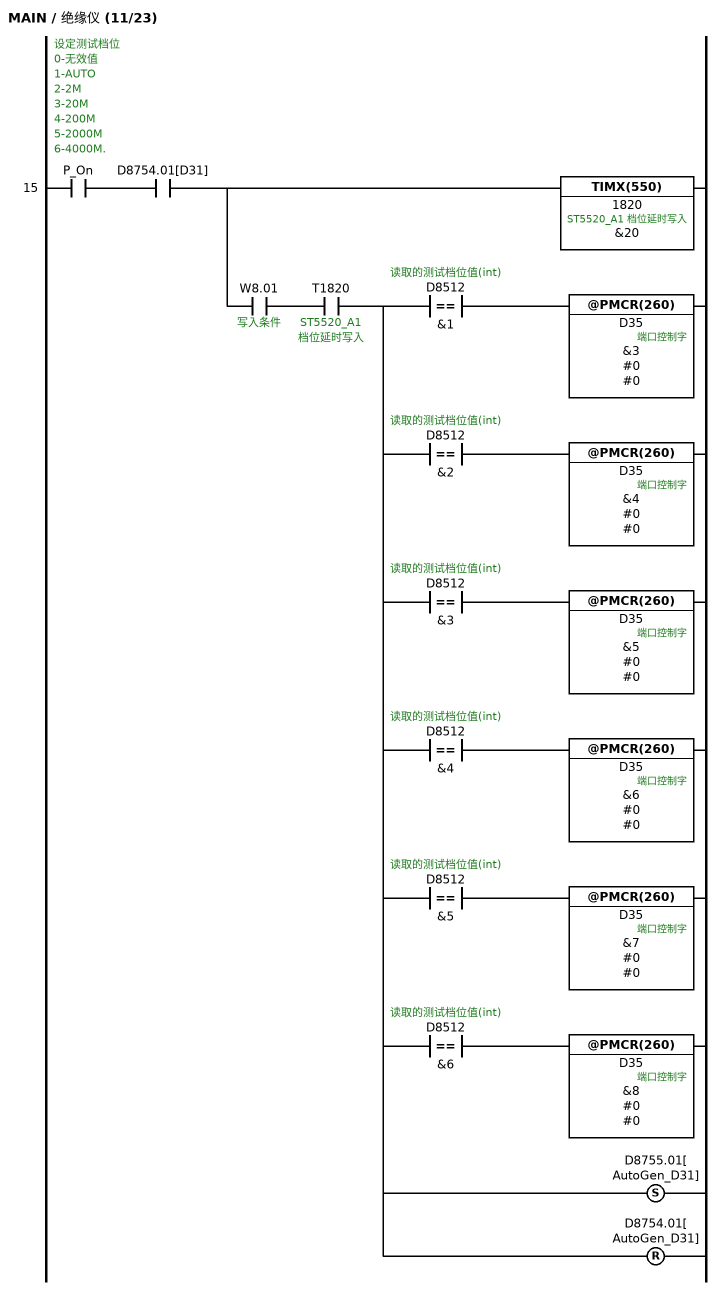
; rung 15: 设定测试档位 / 0-无效值 / 1-AUTO / 2-2M / 3-20M / 4-200M / 5-2000M / 6-4000M.
LD P_On
AND D8754.01[D31]
TIMX(550) 1820 &20  ; ST5520_A1 档位延时写入
AND W8.01  ; 写入条件
AND T1820  ; ST5520_A1 档位延时写入
OUT TR0
AND=(300) D8512 &1  ; 读取的测试档位值(int)
@PMCR(260) D35 &3 #0 #0  ; 端口控制字
LD TR0
AND=(300) D8512 &2  ; 读取的测试档位值(int)
@PMCR(260) D35 &4 #0 #0  ; 端口控制字
LD TR0
AND=(300) D8512 &3  ; 读取的测试档位值(int)
@PMCR(260) D35 &5 #0 #0  ; 端口控制字
LD TR0
AND=(300) D8512 &4  ; 读取的测试档位值(int)
@PMCR(260) D35 &6 #0 #0  ; 端口控制字
LD TR0
AND=(300) D8512 &5  ; 读取的测试档位值(int)
@PMCR(260) D35 &7 #0 #0  ; 端口控制字
LD TR0
AND=(300) D8512 &6  ; 读取的测试档位值(int)
@PMCR(260) D35 &8 #0 #0  ; 端口控制字
LD TR0
SET D8755.01[AutoGen_D31]
RSET D8754.01[AutoGen_D31]

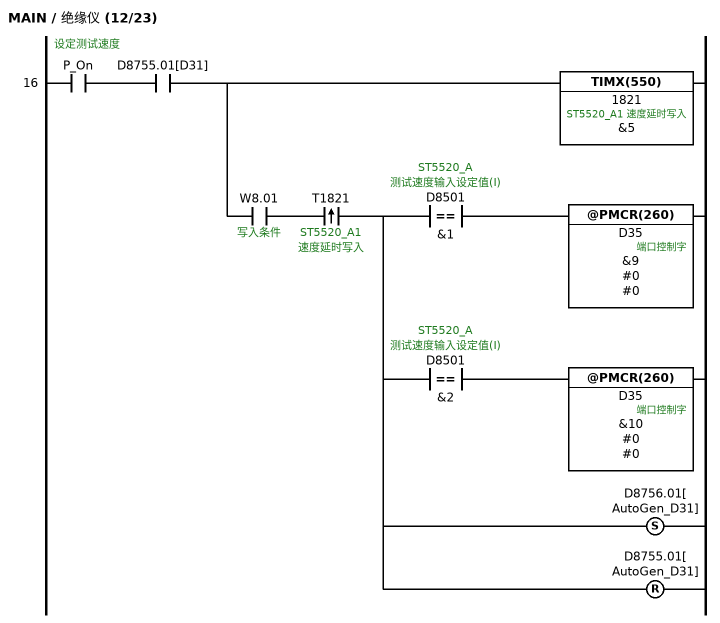
; rung 16: 设定测试速度
LD P_On
AND D8755.01[D31]
TIMX(550) 1821 &5  ; ST5520_A1 速度延时写入
AND W8.01  ; 写入条件
@AND T1821  ; ST5520_A1 速度延时写入
OUT TR0
AND=(300) D8501 &1  ; ST5520_A 测试速度输入设定值(I)
@PMCR(260) D35 &9 #0 #0  ; 端口控制字
LD TR0
AND=(300) D8501 &2  ; ST5520_A 测试速度输入设定值(I)
@PMCR(260) D35 &10 #0 #0  ; 端口控制字
LD TR0
SET D8756.01[AutoGen_D31]
RSET D8755.01[AutoGen_D31]

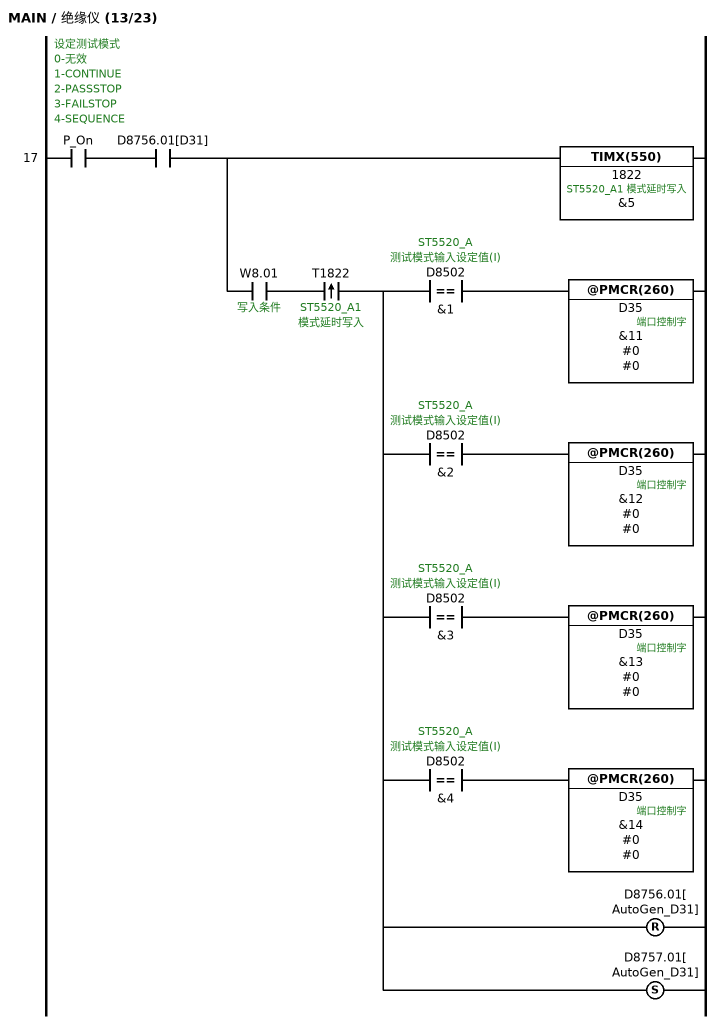
; rung 17: 设定测试模式 / 0-无效 / 1-CONTINUE / 2-PASSSTOP / 3-FAILSTOP / 4-SEQUENCE
LD P_On
AND D8756.01[D31]
TIMX(550) 1822 &5  ; ST5520_A1 模式延时写入
AND W8.01  ; 写入条件
@AND T1822  ; ST5520_A1 模式延时写入
OUT TR0
AND=(300) D8502 &1  ; ST5520_A 测试模式输入设定值(I)
@PMCR(260) D35 &11 #0 #0  ; 端口控制字
LD TR0
AND=(300) D8502 &2  ; ST5520_A 测试模式输入设定值(I)
@PMCR(260) D35 &12 #0 #0  ; 端口控制字
LD TR0
AND=(300) D8502 &3  ; ST5520_A 测试模式输入设定值(I)
@PMCR(260) D35 &13 #0 #0  ; 端口控制字
LD TR0
AND=(300) D8502 &4  ; ST5520_A 测试模式输入设定值(I)
@PMCR(260) D35 &14 #0 #0  ; 端口控制字
LD TR0
RSET D8756.01[AutoGen_D31]
SET D8757.01[AutoGen_D31]

